// TIA Portal V20 export
TYPE "IO_DO"
   STRUCT
      OUT : Struct
         Output : Bool;
      END_STRUCT;
   END_STRUCT;
END_TYPE
